Fanuc KAREL source: V_CLR_VAMAP.kl

PROGRAM T
%NOLOCKGROUP
VAR
 v0 : STRING[40]
 v1 : INTEGER
BEGIN
 V_CLR_VAMAP(v0, v1)
END T
